{attribute 'qualified_only'}
VAR_GLOBAL	
	S1 AT %I*: BOOL;	// Taster (1) (Schliesser)
END_VAR

(* stored: Version 1.1.0.1, ProductVersion 3.1.4024.4
   GVL SimDI: Id {c2d05302-d374-4f85-80dd-41006a3e3277} *)
